{attribute 'reflection'}
FUNCTION_BLOCK FB_LAMP_DIMM IMPLEMENTS I_LampCtrl
VAR_INPUT
END_VAR
VAR_OUTPUT
END_VAR
VAR
	
	fOut :REAL;
	fInc :REAL:=0.5;
	iOutHw AT%Q*:INT; // Output to Dimmer
	
	{attribute 'instance-path'}
	{attribute 'no_init'}
	sPath: STRING;
END_VAR

METHOD OFF : BOOL
// implementation dimm++. 
//Intensity in 0..100%  variable fOut 
fOut :=fOut - fInc;
IF fOut < 0.0 THEN
    fOut :=0.0;
	OFF := TRUE;
ELSE
	OFF := FALSE;
END_IF

// conversion to hardware output 0..32767
iOutHw := LIMIT (0,REAL_TO_INT(fOut * 32.767),32767); // for dimmer output
END_METHOD

METHOD ON : BOOL
// implementation dimm++. 
//Intensity in 0..100%  variable fOut 
fOut :=fOut + fInc;
IF fOut > 100.0 THEN
    fOut :=100.0;
	On := TRUE;
ELSE
	On := FALSE;
END_IF
iOutHw := LIMIT (0,REAL_TO_INT(fOut * 327.67),32767); // for dimmer output
END_METHOD

PROPERTY State : string
GET
State := CONCAT('Object:', sPath); 
State := CONCAT(State, 'State (%):'); 
State := CONCAT(State, REAL_TO_STRING(fOut));
END_GET
END_PROPERTY

END_FUNCTION_BLOCK

(* stored: Version 1.1.0.1, ProductVersion 3.1.4024.6
   POU FB_LAMP_DIMM: Id {3a1eccb9-1d45-4250-a7a3-681ecb969535}, SpecialFunc None
   Method OFF: Id {4aa2126f-d62e-44be-9e00-c24d7e832071}
   Method ON: Id {ff6a5352-1f91-4bf4-9a0c-06c368dd320b}
   Property State: Id {5ac3d078-2cca-47c3-aad2-7982bc0c6545}
   Get Get: Id {f1143ca4-13ea-4d9b-b180-40fbefa4adc8} *)
